// Test-only access to state, timer and permissive internals for isolated cases.
// The cyclic body supplies one synthetic active-step observation before SUPER^()
// because transition unit tests do not run a complete application scan.
// Coverage regressions use real FB_StateMachine instances instead of this probe.
// Plain VAR members are accessible to TwinCAT subclasses. This type is excluded
// from the shipped library.
FUNCTION_BLOCK FB_StateMachine_Probe EXTENDS TcForge.FB_StateMachine

// Transition unit tests supply no full application scan. Coverage is tested with real FB_StateMachine instances.
_activeStepCalls := 1;
SUPER^();

// Full isolation reset for the shared suite-level probe. Clears fault
// book-keeping, command-request flags, permissive / interlock live
// state, rising-edge memory on the SM's internal triggers, and
// published Status back to its power-on values. Each test method
// calls this in its own Setup() so tests see a clean slate even
// though the probe instance itself is reused.
//
METHOD PUBLIC ResetAll
VAR
    i : UDINT;
END_VAR
_ClearFault();
_stepFailurePending := FALSE;
_stepRecoveryPending := FALSE;
_coverageStep := -1;
_activeStepCalls := 0;
Status.ShutdownFailed := FALSE;
Status.FailedStep := 0;
inpShutdownConfirmed := FALSE;
bSourceLockedToProg := FALSE;
Status.AtRecoveryStep := FALSE;
inpSubmoduleFaulted := FALSE;

_abortRequested         := FALSE;
_completeStateRequested := FALSE;
_homeRequested          := FALSE;
_pauseRequested         := FALSE;
_proceedRequested       := FALSE;
_startRequested         := FALSE;
_stopRequested          := FALSE;
_retryActive            := FALSE;
RetryComplete           := FALSE;
_blockedCode            := 0;
_starvedCode            := 0;

// Order matters for FB_Interlock: Reset() snaps _latchedBits to the
// current nLiveBits, so the live bits must already be good before the
// reset. Otherwise a bit left FALSE by a previous test (e.g. the
// running-interlock-trip case) stays latched bad across the reset and
// makes every subsequent test look like the interlock auto-aborted.
// FB_Permissives is non-latching so the order doesn't matter there,
// but we keep it consistent.
FOR i := 0 TO 63 DO
    permHome.MapInput(bitIndex := i, inputValue := TRUE);
    permStart.MapInput(bitIndex := i, inputValue := TRUE);
    permProceed.MapInput(bitIndex := i, inputValue := TRUE);
    permAuto.MapInput(bitIndex := i, inputValue := TRUE);
    intlkRunning.MapInput(bitIndex := i, inputValue := TRUE);
END_FOR;
cfgAutoRun := FALSE;
StepTimer(IN := FALSE);
permHome.Reset();
permStart.Reset();
permProceed.Reset();
permAuto.Reset();
intlkRunning.Reset();

R_TRIG_1(CLK := FALSE);

Status.State            := TcForge.E_SM_State.STOPPED;
Status.LastState        := TcForge.E_SM_State.STOPPED;
Status.Step.Current     := 0;
Status.Step.Next        := 0;
Status.Step.TimerSeconds := 0.0;
Status.Faulted          := FALSE;
Status.SubmoduleFaulted := FALSE;
Status.BlockedCondition := 0;
Status.StarvedCondition := 0;
Status.AutoCycleRequest := FALSE;

_nextStep      := 0;
_returnState   := TcForge.E_SM_State.STOPPED;
ReturnNextStep := 0;
PreviousStep   := 0;
END_METHOD

// Force the active step number. Lets FB_Step see _active = TRUE without
// us having to drive Home/Start/state transitions end-to-end.
METHOD PUBLIC SetCurrentStep
VAR_INPUT
    nStep : DINT;
END_VAR
Status.Step.Current := nStep;
END_METHOD

// Inject a step-timer reading so timeout branches can be tested without
// actually letting wall-clock time pass. The production SM owns the
// timer — here we just write the published value directly.
METHOD PUBLIC SetTimerSeconds
VAR_INPUT
    seconds : REAL;
END_VAR
Status.Step.TimerSeconds := seconds;
END_METHOD

// Park the SM in a specific state without walking the full
// Home/Start/Complete command sequence. Used by the transition tests
// to set up "machine is in state X, now issue command Y" without
// running a sequence first.
METHOD PUBLIC ForceState
VAR_INPUT
    state : TcForge.E_SM_State;
END_VAR
Status.State := state;
END_METHOD

// Set Status.LastState directly. Needed for the AutoCycle path
// (fires when State=READY AND LastState=RUNNING) without walking
// a full RUNNING -> READY transition first.
METHOD PUBLIC ForceLastState
VAR_INPUT
    state : TcForge.E_SM_State;
END_VAR
Status.LastState := state;
END_METHOD

// Drive _nextStep directly. Used with ForceState+SetCurrentStep to
// simulate "mid-sequence" — if _nextStep stays at 0 while a forced
// Current lands inside the state's step range, R_TRIG_5 fires a
// spurious sequence-complete that tests don't want.
METHOD PUBLIC ForceNextStep
VAR_INPUT
    nStep : DINT;
END_VAR
_nextStep := nStep;
END_METHOD

// Map a bit into the private permHome block so the Home-permissive
// gate can be observed. Without this the internal FB_Permissives has
// no external mapping surface on the SM, and every test would see
// "all perms OK" by default.
METHOD PUBLIC MapHomePerm
VAR_INPUT
    bitIndex : UDINT;
    bGood    : BOOL;
END_VAR
permHome.MapInput(bitIndex := bitIndex, inputValue := bGood);
END_METHOD

METHOD PUBLIC MapStartPerm
VAR_INPUT
    bitIndex : UDINT;
    bGood    : BOOL;
END_VAR
permStart.MapInput(bitIndex := bitIndex, inputValue := bGood);
END_METHOD

METHOD PUBLIC MapProceedPerm
VAR_INPUT
    bitIndex : UDINT;
    bGood    : BOOL;
END_VAR
permProceed.MapInput(bitIndex := bitIndex, inputValue := bGood);
END_METHOD

METHOD PUBLIC MapAutoPerm
VAR_INPUT
    bitIndex : UDINT;
    bGood    : BOOL;
END_VAR
permAuto.MapInput(bitIndex := bitIndex, inputValue := bGood);
END_METHOD

END_FUNCTION_BLOCK

(* stored: Version 1.1.0.1, ProductVersion 3.1.4026.12
   POU FB_StateMachine_Probe: Id {c3d4e5f6-a7b8-9012-cdef-000000001100}, SpecialFunc None
   Method ResetAll: Id {c3d4e5f6-a7b8-9012-cdef-000000001198}
   Method SetCurrentStep: Id {c3d4e5f6-a7b8-9012-cdef-000000001101}
   Method SetTimerSeconds: Id {c3d4e5f6-a7b8-9012-cdef-000000001102}
   Method ForceState: Id {c3d4e5f6-a7b8-9012-cdef-000000001103}
   Method ForceLastState: Id {c3d4e5f6-a7b8-9012-cdef-000000001104}
   Method ForceNextStep: Id {c3d4e5f6-a7b8-9012-cdef-000000001105}
   Method MapHomePerm: Id {c3d4e5f6-a7b8-9012-cdef-000000001106}
   Method MapStartPerm: Id {c3d4e5f6-a7b8-9012-cdef-000000001107}
   Method MapProceedPerm: Id {c3d4e5f6-a7b8-9012-cdef-000000001108}
   Method MapAutoPerm: Id {c3d4e5f6-a7b8-9012-cdef-000000001109} *)
